(* 
| :Description: this function block is the Contactor FeedbackNO + thermal relay connect toghther.
| Then wiring have to series by Digital output to NC thermal relay to Coil
*)
FUNCTION_BLOCK FB_Contactor1FB_ThermalRelay EXTENDS FB_ContactorFBNO IMPLEMENTS I_ActivePower

VAR
	piFR		: FB_DigitalInput;// thermal relay NO
	bOverload	: BOOL;
END_VAR

bOverload :=  piFR.In;
SUPER^();

PROPERTY IsOverload : REFERENCE to bool
GET
isOverload ref= bOverload;
END_GET
END_PROPERTY

PROPERTY ReasonError : string
GET
IF isOverload THEN 
	ReasonError := 'ThermalRelay OverLoad';
ELSE
	ReasonError := 'Coil of Contactor or NO contact work incorrectly';
END_IF
END_GET
END_PROPERTY

PROPERTY Ref_piFR : reference to FB_DigitalInput
GET
Ref_piFR ref= piFR;
END_GET
END_PROPERTY

END_FUNCTION_BLOCK

(* stored: Version 1.1.0.1, ProductVersion 3.1.4024.12
   POU FB_Contactor1FB_ThermalRelay: Id {8da0f9a8-4739-4828-afed-8042b6912c75}, SpecialFunc None
   Property IsOverload: Id {3ef34ec1-df4f-4a8a-961a-01f509836c97}
   Get Get: Id {658399c6-726c-4361-baf2-50ffc815893c}
   Property ReasonError: Id {f7227d89-79e3-4423-896e-d3d00113b065}
   Get Get: Id {3716ab08-388e-43f1-a049-6a26dd1d46b4}
   Property Ref_piFR: Id {ebfc3958-0b40-4bbd-8074-bd0772026004}
   Get Get: Id {c07d0155-7008-4de9-b594-2b395f284b5b} *)
